LIN {X 0,Y 103.951,Z 742.341,A -85,B 0,C 180,E1 -28115.783,E2 -28115.783} C_VEL
LIN {X 0,Y 96.349,Z 750.933,A -85,B 0,C 180,E1 -28120.019,E2 -28120.019} C_VEL
LIN {X 0,Y 88.516,Z 758.718,A -85,B 0,C 180,E1 -28125.825,E2 -28125.825} C_VEL
LIN {X 0,Y 83.316,Z 763.333,A -85,B 0,C 180,E1 -28130.76,E2 -28130.76} C_VEL
LIN {X 0,Y 78.062,Z 767.663,A -85,B 0,C 180,E1 -28137.31,E2 -28137.31} C_VEL
LIN {X 0,Y 75.138,Z 769.96,A -85,B 0,C 180,E1 -28142.122,E2 -28142.122} C_VEL
LIN {X 0,Y 72.891,Z 771.823,A -85,B 0,C 180,E1 -28147.32,E2 -28147.32} C_VEL
LIN {X 0,Y 70.141,Z 774.222,A -85,B 0,C 180,E1 -28158.445,E2 -28158.445} C_VEL
LIN {X 0,Y 69.62,Z 774.834,A -85,B 0,C 180,E1 -28164.212,E2 -28164.212} C_VEL
LIN {X 0,Y 69.698,Z 775.05,A -85,B 0,C 180,E1 -28170.005,E2 -28170.005} C_VEL
LIN {X 0,Y 70.018,Z 774.825,A -85,B 0,C 180,E1 -28175.766,E2 -28175.766} C_VEL
LIN {X 0,Y 72.328,Z 773.205,A -85,B 0,C 180,E1 -28186.953,E2 -28186.953} C_VEL
LIN {X 0,Y 74.422,Z 771.801,A -85,B 0,C 180,E1 -28192.199,E2 -28192.199} C_VEL
LIN {X 0,Y 78.894,Z 768.873,A -85,B 0,C 180,E1 -28199.342,E2 -28199.342} C_VEL
LIN {X 0,Y 84.664,Z 764.918,A -85,B 0,C 180,E1 -28205.531,E2 -28205.531} C_VEL
LIN {X 0,Y 91.748,Z 759.838,A -85,B 0,C 180,E1 -28210.63,E2 -28210.63} C_VEL
LIN {X 0,Y 97.262,Z 756.003,A -85,B 0,C 180,E1 -28213.358,E2 -28213.358} C_VEL
LIN {X 0,Y 98.436,Z 756.44,A -85,B 0,C 180,E1 -28214.122,E2 -28214.122} C_VEL
LIN {X 0,Y 99.632,Z 757.554,A -85,B 0,C 180,E1 -28215.138,E2 -28215.138} C_VEL
LIN {X 0,Y 98.401,Z 756.23,A -85,B 0,C 180,E1 -28217.273,E2 -28217.273} C_VEL
LIN {X 0,Y 94.133,Z 751.514,A -85,B 0,C 180,E1 -28221.297,E2 -28221.297} C_VEL
LIN {X 0,Y 92.534,Z 750.794,A -85,B 0,C 180,E1 -28222.584,E2 -28222.584} C_VEL
LIN {X 0,Y 89.015,Z 750.077,A -85,B 0,C 180,E1 -28226.45,E2 -28226.45} C_VEL
LIN {X 0,Y 86.882,Z 747.385,A -85,B 0,C 180,E1 -28232.857,E2 -28232.857} C_VEL
LIN {X 0,Y 85.307,Z 746.912,A -85,B 0,C 180,E1 -28235.674,E2 -28235.674} C_VEL
LIN {X 0,Y 84.144,Z 745.468,A -85,B 0,C 180,E1 -28240.483,E2 -28240.483} C_VEL
LIN {X 0,Y 84.612,Z 743,A -85,B 0,C 180,E1 -28245.571,E2 -28245.571} C_VEL
LIN {X 0,Y 85.192,Z 740.288,A -85,B 0,C 180,E1 -28253.587,E2 -28253.587} C_VEL
LIN {X 0,Y 85.413,Z 739.646,A -85,B 0,C 180,E1 -28256.213,E2 -28256.213} C_VEL
LIN {X 0,Y 84.758,Z 739.885,A -85,B 0,C 180,E1 -28260.73,E2 -28260.73} C_VEL
LIN {X 0,Y 84.568,Z 740.192,A -85,B 0,C 180,E1 -28265.315,E2 -28265.315} C_VEL
LIN {X 0,Y 85.486,Z 739.643,A -85,B 0,C 180,E1 -28267.912,E2 -28267.912} C_VEL
LIN {X 0,Y 88.337,Z 737.785,A -85,B 0,C 180,E1 -28271.763,E2 -28271.763} C_VEL
LIN {X 0,Y 90.112,Z 736.61,A -85,B 0,C 180,E1 -28273.531,E2 -28273.531} C_VEL
LIN {X 0,Y 92.574,Z 734.85,A -85,B 0,C 180,E1 -28275.41,E2 -28275.41} C_VEL
LIN {X 0,Y 97.676,Z 731.683,A -85,B 0,C 180,E1 -28279.541,E2 -28279.541} C_VEL
LIN {X 0,Y 102.495,Z 728.307,A -85,B 0,C 180,E1 -28282.156,E2 -28282.156} C_VEL
LIN {X 0,Y 111.157,Z 722.092,A -85,B 0,C 180,E1 -28286.269,E2 -28286.269} C_VEL
LIN {X 0,Y 113.724,Z 720.096,A -85,B 0,C 180,E1 -28287.244,E2 -28287.244} C_VEL
LIN {X 0,Y 113.59,Z 721.326,A -85,B 0,C 180,E1 -28288.149,E2 -28288.149} C_VEL
LIN {X 0,Y 106.442,Z 731.795,A -85,B 0,C 180,E1 -28290.863,E2 -28290.863} C_VEL
LIN {X 0,Y 99.593,Z 740.264,A -85,B 0,C 180,E1 -28293.983,E2 -28293.983} C_VEL
LIN {X 0,Y 91.701,Z 748.632,A -85,B 0,C 180,E1 -28298.418,E2 -28298.418} C_VEL
LIN {X 0,Y 85.822,Z 754.124,A -85,B 0,C 180,E1 -28302.517,E2 -28302.517} C_VEL
LIN {X 0,Y 79.072,Z 759.618,A -85,B 0,C 180,E1 -28308.189,E2 -28308.189} C_VEL
LIN {X 0,Y 73.326,Z 763.919,A -85,B 0,C 180,E1 -28314.889,E2 -28314.889} C_VEL
LIN {X 0,Y 70.064,Z 766.192,A -85,B 0,C 180,E1 -28319.892,E2 -28319.892} C_VEL
LIN {X 0,Y 67.35,Z 768.037,A -85,B 0,C 180,E1 -28325.324,E2 -28325.324} C_VEL
LIN {X 0,Y 65.246,Z 769.422,A -85,B 0,C 180,E1 -28331.141,E2 -28331.141} C_VEL
LIN {X 0,Y 62.947,Z 771.009,A -85,B 0,C 180,E1 -28343.584,E2 -28343.584} C_VEL
LIN {X 0,Y 62.722,Z 771.232,A -85,B 0,C 180,E1 -28349.994,E2 -28349.994} C_VEL
LIN {X 0,Y 62.94,Z 771.037,A -85,B 0,C 180,E1 -28356.405,E2 -28356.405} C_VEL
LIN {X 0,Y 65.24,Z 769.487,A -85,B 0,C 180,E1 -28368.849,E2 -28368.849} C_VEL
LIN {X 0,Y 67.334,Z 768.13,A -85,B 0,C 180,E1 -28374.671,E2 -28374.671} C_VEL
LIN {X 0,Y 71.588,Z 765.258,A -85,B 0,C 180,E1 -28382.674,E2 -28382.674} C_VEL
LIN {X 0,Y 76.942,Z 761.361,A -85,B 0,C 180,E1 -28389.74,E2 -28389.74} C_VEL
LIN {X 0,Y 83.405,Z 756.332,A -85,B 0,C 180,E1 -28395.738,E2 -28395.738} C_VEL
LIN {X 0,Y 90.529,Z 749.996,A -85,B 0,C 180,E1 -28400.918,E2 -28400.918} C_VEL
LIN {X 0,Y 97.95,Z 742.366,A -85,B 0,C 180,E1 -28405.233,E2 -28405.233} C_VEL
LIN {X 0,Y 104.986,Z 733.989,A -85,B 0,C 180,E1 -28408.589,E2 -28408.589} C_VEL
LIN {X 0,Y 112.075,Z 724.121,A -85,B 0,C 180,E1 -28411.384,E2 -28411.384} C_VEL
LIN {X 0,Y 118.662,Z 713.001,A -85,B 0,C 180,E1 -28413.604,E2 -28413.604} C_VEL
LIN {X 0,Y 123.869,Z 702.096,A -85,B 0,C 180,E1 -28415.194,E2 -28415.194} C_VEL
LIN {X 0,Y 128.403,Z 690.023,A -85,B 0,C 180,E1 -28416.453,E2 -28416.453} C_VEL
LIN {X 0,Y 131.881,Z 677.141,A -85,B 0,C 180,E1 -28417.41,E2 -28417.41} C_VEL
LIN {X 0,Y 134.056,Z 664.506,A -85,B 0,C 180,E1 -28418.006,E2 -28418.006} C_VEL
LIN {X 0,Y 134.924,Z 656.338,A -85,B 0,C 180,E1 -28418.309,E2 -28418.309} C_VEL
LIN {X 0,Y 132.782,Z 650.972,A -85,B 0,C 180,E1 -28421.683,E2 -28421.683} C_VEL
LIN {X 0,Y 131.13,Z 647.298,A -85,B 0,C 180,E1 -28424.778,E2 -28424.778} C_VEL
LIN {X 0,Y 129.8,Z 644.377,A -85,B 0,C 180,E1 -28427.888,E2 -28427.888} C_VEL
LIN {X 0,Y 128.772,Z 641.836,A -85,B 0,C 180,E1 -28431.17,E2 -28431.17} C_VEL
LIN {X 0,Y 127.754,Z 638.207,A -85,B 0,C 180,E1 -28440,E2 -28440} C_VEL
LIN {X 0,Y 128.97,Z 642.375,A -85,B 0,C 180,E1 -28449.211,E2 -28449.211} C_VEL
LIN {X 0,Y 130.645,Z 646.22,A -85,B 0,C 180,E1 -28453.811,E2 -28453.811} C_VEL
LIN {X 0,Y 132.545,Z 650.385,A -85,B 0,C 180,E1 -28457.537,E2 -28457.537} C_VEL
LIN {X 0,Y 133.588,Z 653.257,A -85,B 0,C 180,E1 -28459.346,E2 -28459.346} C_VEL
LIN {X 0,Y 134.794,Z 657.853,A -85,B 0,C 180,E1 -28461.406,E2 -28461.406} C_VEL
LIN {X 0,Y 132.887,Z 673.229,A -85,B 0,C 180,E1 -28461.953,E2 -28461.953} C_VEL
LIN {X 0,Y 129.998,Z 686.389,A -85,B 0,C 180,E1 -28462.692,E2 -28462.692} C_VEL
LIN {X 0,Y 125.715,Z 699.337,A -85,B 0,C 180,E1 -28463.741,E2 -28463.741} C_VEL
LIN {X 0,Y 120.339,Z 711.572,A -85,B 0,C 180,E1 -28465.154,E2 -28465.154} C_VEL
LIN {X 0,Y 114.322,Z 722.478,A -85,B 0,C 180,E1 -28466.959,E2 -28466.959} C_VEL
LIN {X 0,Y 107.009,Z 733.323,A -85,B 0,C 180,E1 -28469.524,E2 -28469.524} C_VEL
LIN {X 0,Y 99.949,Z 742.138,A -85,B 0,C 180,E1 -28472.465,E2 -28472.465} C_VEL
LIN {X 0,Y 91.931,Z 750.73,A -85,B 0,C 180,E1 -28476.617,E2 -28476.617} C_VEL
LIN {X 0,Y 84.142,Z 757.985,A -85,B 0,C 180,E1 -28481.928,E2 -28481.928} C_VEL
LIN {X 0,Y 77.939,Z 763.129,A -85,B 0,C 180,E1 -28487.452,E2 -28487.452} C_VEL
LIN {X 0,Y 72.171,Z 767.458,A -85,B 0,C 180,E1 -28494.254,E2 -28494.254} C_VEL
LIN {X 0,Y 68.92,Z 769.755,A -85,B 0,C 180,E1 -28499.351,E2 -28499.351} C_VEL
LIN {X 0,Y 66.352,Z 771.617,A -85,B 0,C 180,E1 -28504.939,E2 -28504.939} C_VEL
LIN {X 0,Y 64.452,Z 773.016,A -85,B 0,C 180,E1 -28510.912,E2 -28510.912} C_VEL
LIN {X 0,Y 63.176,Z 774.017,A -85,B 0,C 180,E1 -28517.151,E2 -28517.151} C_VEL
LIN {X 0,Y 62.555,Z 774.629,A -85,B 0,C 180,E1 -28523.555,E2 -28523.555} C_VEL
LIN {X 0,Y 62.607,Z 774.846,A -85,B 0,C 180,E1 -28530.006,E2 -28530.006} C_VEL
LIN {X 0,Y 62.958,Z 774.62,A -85,B 0,C 180,E1 -28536.415,E2 -28536.415} C_VEL
LIN {X 0,Y 65.591,Z 773.001,A -85,B 0,C 180,E1 -28548.756,E2 -28548.756} C_VEL
LIN {X 0,Y 67.928,Z 771.596,A -85,B 0,C 180,E1 -28554.453,E2 -28554.453} C_VEL
LIN {X 0,Y 72.809,Z 768.668,A -85,B 0,C 180,E1 -28562.071,E2 -28562.071} C_VEL
LIN {X 0,Y 79.017,Z 764.713,A -85,B 0,C 180,E1 -28568.512,E2 -28568.512} C_VEL
LIN {X 0,Y 86.479,Z 759.632,A -85,B 0,C 180,E1 -28573.697,E2 -28573.697} C_VEL
LIN {X 0,Y 91.24,Z 756.158,A -85,B 0,C 180,E1 -28576.112,E2 -28576.112} C_VEL
LIN {X 0,Y 87.932,Z 754.779,A -85,B 0,C 180,E1 -28580.253,E2 -28580.253} C_VEL
LIN {X 0,Y 84.169,Z 754.131,A -85,B 0,C 180,E1 -28584.233,E2 -28584.233} C_VEL
LIN {X 0,Y 80.136,Z 751.193,A -85,B 0,C 180,E1 -28593.992,E2 -28593.992} C_VEL
LIN {X 0,Y 78.65,Z 749.984,A -85,B 0,C 180,E1 -28599.058,E2 -28599.058} C_VEL
LIN {X 0,Y 79.024,Z 746.684,A -85,B 0,C 180,E1 -28608.06,E2 -28608.06} C_VEL
LIN {X 0,Y 83.57,Z 741.075,A -85,B 0,C 180,E1 -28624.824,E2 -28624.824} C_VEL
LIN {X 0,Y 85.486,Z 739.643,A -85,B 0,C 180,E1 -28627.912,E2 -28627.912} C_VEL
LIN {X 0,Y 87.027,Z 738.869,A -85,B 0,C 180,E1 -28631.283,E2 -28631.283} C_VEL
LIN {X 0,Y 90.368,Z 738.328,A -85,B 0,C 180,E1 -28638.799,E2 -28638.799} C_VEL
LIN {X 0,Y 92.458,Z 737.403,A -85,B 0,C 180,E1 -28640.822,E2 -28640.822} C_VEL
LIN {X 0,Y 96.855,Z 734.883,A -85,B 0,C 180,E1 -28643.522,E2 -28643.522} C_VEL
LIN {X 0,Y 103.773,Z 730.418,A -85,B 0,C 180,E1 -28646.551,E2 -28646.551} C_VEL
LIN {X 0,Y 102.975,Z 732.004,A -85,B 0,C 180,E1 -28647.464,E2 -28647.464} C_VEL
LIN {X 0,Y 95.662,Z 740.618,A -85,B 0,C 180,E1 -28650.519,E2 -28650.519} C_VEL
LIN {X 0,Y 88.192,Z 748.173,A -85,B 0,C 180,E1 -28654.361,E2 -28654.361} C_VEL
LIN {X 0,Y 81.191,Z 754.331,A -85,B 0,C 180,E1 -28658.82,E2 -28658.82} C_VEL
LIN {X 0,Y 73.933,Z 759.824,A -85,B 0,C 180,E1 -28664.519,E2 -28664.519} C_VEL
LIN {X 0,Y 67.626,Z 764.125,A -85,B 0,C 180,E1 -28671.418,E2 -28671.418} C_VEL
LIN {X 0,Y 64.009,Z 766.398,A -85,B 0,C 180,E1 -28676.696,E2 -28676.696} C_VEL
LIN {X 0,Y 60.978,Z 768.242,A -85,B 0,C 180,E1 -28682.541,E2 -28682.541} C_VEL
LIN {X 0,Y 58.576,Z 769.627,A -85,B 0,C 180,E1 -28688.897,E2 -28688.897} C_VEL
LIN {X 0,Y 55.914,Z 771.214,A -85,B 0,C 180,E1 -28702.773,E2 -28702.773} C_VEL
LIN {X 0,Y 55.649,Z 771.436,A -85,B 0,C 180,E1 -28709.993,E2 -28709.993} C_VEL
LIN {X 0,Y 55.908,Z 771.241,A -85,B 0,C 180,E1 -28717.215,E2 -28717.215} C_VEL
LIN {X 0,Y 58.569,Z 769.691,A -85,B 0,C 180,E1 -28731.092,E2 -28731.092} C_VEL
LIN {X 0,Y 60.961,Z 768.334,A -85,B 0,C 180,E1 -28737.454,E2 -28737.454} C_VEL
LIN {X 0,Y 65.72,Z 765.462,A -85,B 0,C 180,E1 -28746.019,E2 -28746.019} C_VEL
LIN {X 0,Y 71.623,Z 761.565,A -85,B 0,C 180,E1 -28753.376,E2 -28753.376} C_VEL
LIN {X 0,Y 78.616,Z 756.535,A -85,B 0,C 180,E1 -28759.445,E2 -28759.445} C_VEL
LIN {X 0,Y 86.231,Z 750.199,A -85,B 0,C 180,E1 -28764.582,E2 -28764.582} C_VEL
LIN {X 0,Y 94.363,Z 742.273,A -85,B 0,C 180,E1 -28768.918,E2 -28768.918} C_VEL
LIN {X 0,Y 102.93,Z 732.412,A -85,B 0,C 180,E1 -28772.569,E2 -28772.569} C_VEL
LIN {X 0,Y 110.366,Z 722.044,A -85,B 0,C 180,E1 -28775.143,E2 -28775.143} C_VEL
LIN {X 0,Y 117.211,Z 710.357,A -85,B 0,C 180,E1 -28777.195,E2 -28777.195} C_VEL
LIN {X 0,Y 122.573,Z 698.847,A -85,B 0,C 180,E1 -28778.591,E2 -28778.591} C_VEL
LIN {X 0,Y 126.995,Z 686.165,A -85,B 0,C 180,E1 -28779.743,E2 -28779.743} C_VEL
LIN {X 0,Y 130.237,Z 673.11,A -85,B 0,C 180,E1 -28780.514,E2 -28780.514} C_VEL
LIN {X 0,Y 132.088,Z 659.976,A -85,B 0,C 180,E1 -28781.072,E2 -28781.072} C_VEL
LIN {X 0,Y 130.016,Z 654.54,A -85,B 0,C 180,E1 -28785.097,E2 -28785.097} C_VEL
LIN {X 0,Y 128.555,Z 651.088,A -85,B 0,C 180,E1 -28788.769,E2 -28788.769} C_VEL
LIN {X 0,Y 127.631,Z 648.651,A -85,B 0,C 180,E1 -28792.087,E2 -28792.087} C_VEL
LIN {X 0,Y 126.869,Z 645.407,A -85,B 0,C 180,E1 -28800,E2 -28800} C_VEL
LIN {X 0,Y 127.846,Z 649.203,A -85,B 0,C 180,E1 -28808.437,E2 -28808.437} C_VEL
LIN {X 0,Y 129.208,Z 652.693,A -85,B 0,C 180,E1 -28812.666,E2 -28812.666} C_VEL
LIN {X 0,Y 130.912,Z 656.842,A -85,B 0,C 180,E1 -28816.407,E2 -28816.407} C_VEL
LIN {X 0,Y 131.779,Z 659.786,A -85,B 0,C 180,E1 -28818.135,E2 -28818.135} C_VEL
LIN {X 0,Y 132.019,Z 660.871,A -85,B 0,C 180,E1 -28818.627,E2 -28818.627} C_VEL
LIN {X 0,Y 129.975,Z 675.524,A -85,B 0,C 180,E1 -28819.181,E2 -28819.181} C_VEL
LIN {X 0,Y 127.004,Z 687.602,A -85,B 0,C 180,E1 -28819.836,E2 -28819.836} C_VEL
LIN {X 0,Y 122.977,Z 699.263,A -85,B 0,C 180,E1 -28820.722,E2 -28820.722} C_VEL
LIN {X 0,Y 117.495,Z 711.372,A -85,B 0,C 180,E1 -28822.017,E2 -28822.017} C_VEL
LIN {X 0,Y 111.288,Z 722.278,A -85,B 0,C 180,E1 -28823.704,E2 -28823.704} C_VEL
LIN {X 0,Y 103.691,Z 733.121,A -85,B 0,C 180,E1 -28826.104,E2 -28826.104} C_VEL
LIN {X 0,Y 96.311,Z 741.935,A -85,B 0,C 180,E1 -28828.885,E2 -28828.885} C_VEL
LIN {X 0,Y 87.864,Z 750.526,A -85,B 0,C 180,E1 -28832.883,E2 -28832.883} C_VEL
LIN {X 0,Y 80.011,Z 757.409,A -85,B 0,C 180,E1 -28837.771,E2 -28837.771} C_VEL
LIN {X 0,Y 72.858,Z 762.925,A -85,B 0,C 180,E1 -28843.667,E2 -28843.667} C_VEL
LIN {X 0,Y 66.524,Z 767.254,A -85,B 0,C 180,E1 -28850.67,E2 -28850.67} C_VEL
LIN {X 0,Y 62.9,Z 769.551,A -85,B 0,C 180,E1 -28856.044,E2 -28856.044} C_VEL
LIN {X 0,Y 59.955,Z 771.412,A -85,B 0,C 180,E1 -28862.045,E2 -28862.045} C_VEL
LIN {X 0,Y 57.761,Z 772.811,A -85,B 0,C 180,E1 -28868.598,E2 -28868.598} C_VEL
LIN {X 0,Y 56.265,Z 773.812,A -85,B 0,C 180,E1 -28875.54,E2 -28875.54} C_VEL
LIN {X 0,Y 55.512,Z 774.425,A -85,B 0,C 180,E1 -28882.733,E2 -28882.733} C_VEL
LIN {X 0,Y 55.506,Z 774.641,A -85,B 0,C 180,E1 -28890.007,E2 -28890.007} C_VEL
LIN {X 0,Y 55.927,Z 774.416,A -85,B 0,C 180,E1 -28897.226,E2 -28897.226} C_VEL
LIN {X 0,Y 58.92,Z 772.796,A -85,B 0,C 180,E1 -28910.974,E2 -28910.974} C_VEL
LIN {X 0,Y 61.543,Z 771.391,A -85,B 0,C 180,E1 -28917.186,E2 -28917.186} C_VEL
LIN {X 0,Y 66.904,Z 768.463,A -85,B 0,C 180,E1 -28925.299,E2 -28925.299} C_VEL
LIN {X 0,Y 73.602,Z 764.507,A -85,B 0,C 180,E1 -28931.951,E2 -28931.951} C_VEL
LIN {X 0,Y 82.094,Z 759.017,A -85,B 0,C 180,E1 -28937.455,E2 -28937.455} C_VEL
LIN {X 0,Y 81.907,Z 758.248,A -85,B 0,C 180,E1 -28938.913,E2 -28938.913} C_VEL
LIN {X 0,Y 79.297,Z 757.85,A -85,B 0,C 180,E1 -28941.655,E2 -28941.655} C_VEL
LIN {X 0,Y 73.007,Z 754.1,A -85,B 0,C 180,E1 -28957.353,E2 -28957.353} C_VEL
LIN {X 0,Y 73.257,Z 750.666,A -85,B 0,C 180,E1 -28968.938,E2 -28968.938} C_VEL
LIN {X 0,Y 77.803,Z 745.904,A -85,B 0,C 180,E1 -28985.183,E2 -28985.183} C_VEL
LIN {X 0,Y 84.369,Z 742.026,A -85,B 0,C 180,E1 -28994.472,E2 -28994.472} C_VEL
LIN {X 0,Y 86.619,Z 740.762,A -85,B 0,C 180,E1 -28996.501,E2 -28996.501} C_VEL
LIN {X 0,Y 89.295,Z 739.089,A -85,B 0,C 180,E1 -28998.35,E2 -28998.35} C_VEL
LIN {X 0,Y 92.458,Z 737.403,A -85,B 0,C 180,E1 -29000.822,E2 -29000.822} C_VEL
LIN {X 0,Y 93.19,Z 737.288,A -85,B 0,C 180,E1 -29001.855,E2 -29001.855} C_VEL
LIN {X 0,Y 93.192,Z 738.159,A -85,B 0,C 180,E1 -29003.471,E2 -29003.471} C_VEL
LIN {X 0,Y 92.186,Z 740.039,A -85,B 0,C 180,E1 -29005.254,E2 -29005.254} C_VEL
LIN {X 0,Y 90.512,Z 742.304,A -85,B 0,C 180,E1 -29006.911,E2 -29006.911} C_VEL
LIN {X 0,Y 86.442,Z 746.532,A -85,B 0,C 180,E1 -29009.368,E2 -29009.368} C_VEL
LIN {X 0,Y 79.905,Z 752.231,A -85,B 0,C 180,E1 -29012.928,E2 -29012.928} C_VEL
LIN {X 0,Y 76.543,Z 754.826,A -85,B 0,C 180,E1 -29014.936,E2 -29014.936} C_VEL
LIN {X 0,Y 69.143,Z 760.03,A -85,B 0,C 180,E1 -29020.322,E2 -29020.322} C_VEL
LIN {X 0,Y 62.218,Z 764.331,A -85,B 0,C 180,E1 -29027.325,E2 -29027.325} C_VEL
LIN {X 0,Y 58.202,Z 766.603,A -85,B 0,C 180,E1 -29032.853,E2 -29032.853} C_VEL
LIN {X 0,Y 54.761,Z 768.448,A -85,B 0,C 180,E1 -29039.105,E2 -29039.105} C_VEL
LIN {X 0,Y 50.04,Z 770.816,A -85,B 0,C 180,E1 -29053.679,E2 -29053.679} C_VEL
LIN {X 0,Y 48.878,Z 771.418,A -85,B 0,C 180,E1 -29061.726,E2 -29061.726} C_VEL
LIN {X 0,Y 48.565,Z 771.64,A -85,B 0,C 180,E1 -29069.993,E2 -29069.993} C_VEL
LIN {X 0,Y 48.874,Z 771.445,A -85,B 0,C 180,E1 -29078.26,E2 -29078.26} C_VEL
LIN {X 0,Y 50.037,Z 770.861,A -85,B 0,C 180,E1 -29086.307,E2 -29086.307} C_VEL
LIN {X 0,Y 54.743,Z 768.539,A -85,B 0,C 180,E1 -29100.891,E2 -29100.891} C_VEL
LIN {X 0,Y 60.121,Z 765.666,A -85,B 0,C 180,E1 -29110.003,E2 -29110.003} C_VEL
LIN {X 0,Y 66.641,Z 761.769,A -85,B 0,C 180,E1 -29117.572,E2 -29117.572} C_VEL
LIN {X 0,Y 74.199,Z 756.738,A -85,B 0,C 180,E1 -29123.612,E2 -29123.612} C_VEL
LIN {X 0,Y 82.322,Z 750.401,A -85,B 0,C 180,E1 -29128.609,E2 -29128.609} C_VEL
LIN {X 0,Y 90.9,Z 742.475,A -85,B 0,C 180,E1 -29132.755,E2 -29132.755} C_VEL
LIN {X 0,Y 98.346,Z 734.392,A -85,B 0,C 180,E1 -29135.654,E2 -29135.654} C_VEL
LIN {X 0,Y 106.021,Z 724.523,A -85,B 0,C 180,E1 -29138.121,E2 -29138.121} C_VEL
LIN {X 0,Y 113.075,Z 713.401,A -85,B 0,C 180,E1 -29140.053,E2 -29140.053} C_VEL
LIN {X 0,Y 118.627,Z 702.493,A -85,B 0,C 180,E1 -29141.414,E2 -29141.414} C_VEL
LIN {X 0,Y 123.368,Z 690.583,A -85,B 0,C 180,E1 -29142.483,E2 -29142.483} C_VEL
LIN {X 0,Y 127.027,Z 677.928,A -85,B 0,C 180,E1 -29143.295,E2 -29143.295} C_VEL
LIN {X 0,Y 129.382,Z 665.138,A -85,B 0,C 180,E1 -29143.828,E2 -29143.828} C_VEL
LIN {X 0,Y 129.499,Z 663.904,A -85,B 0,C 180,E1 -29143.937,E2 -29143.937} C_VEL
LIN {X 0,Y 128.047,Z 659.755,A -85,B 0,C 180,E1 -29147.519,E2 -29147.519} C_VEL
LIN {X 0,Y 127.06,Z 657.075,A -85,B 0,C 180,E1 -29150.649,E2 -29150.649} C_VEL
LIN {X 0,Y 126.571,Z 655.511,A -85,B 0,C 180,E1 -29152.823,E2 -29152.823} C_VEL
LIN {X 0,Y 125.989,Z 652.578,A -85,B 0,C 180,E1 -29160,E2 -29160} C_VEL
LIN {X 0,Y 126.735,Z 655.923,A -85,B 0,C 180,E1 -29167.568,E2 -29167.568} C_VEL
LIN {X 0,Y 127.96,Z 659.546,A -85,B 0,C 180,E1 -29171.886,E2 -29171.886} C_VEL
LIN {X 0,Y 129.296,Z 663.177,A -85,B 0,C 180,E1 -29175.164,E2 -29175.164} C_VEL
LIN {X 0,Y 129.547,Z 664.051,A -85,B 0,C 180,E1 -29175.739,E2 -29175.739} C_VEL
LIN {X 0,Y 127.446,Z 677.023,A -85,B 0,C 180,E1 -29176.25,E2 -29176.25} C_VEL
LIN {X 0,Y 123.759,Z 690.696,A -85,B 0,C 180,E1 -29176.989,E2 -29176.989} C_VEL
LIN {X 0,Y 119.007,Z 702.96,A -85,B 0,C 180,E1 -29177.901,E2 -29177.901} C_VEL
LIN {X 0,Y 113.427,Z 714.111,A -85,B 0,C 180,E1 -29179.119,E2 -29179.119} C_VEL
LIN {X 0,Y 106.259,Z 725.604,A -85,B 0,C 180,E1 -29180.907,E2 -29180.907} C_VEL
LIN {X 0,Y 99.202,Z 734.859,A -85,B 0,C 180,E1 -29182.94,E2 -29182.94} C_VEL
LIN {X 0,Y 90.072,Z 744.795,A -85,B 0,C 180,E1 -29186.204,E2 -29186.204} C_VEL
LIN {X 0,Y 81.359,Z 752.797,A -85,B 0,C 180,E1 -29190.26,E2 -29190.26} C_VEL
LIN {X 0,Y 72.509,Z 759.682,A -85,B 0,C 180,E1 -29195.787,E2 -29195.787} C_VEL
LIN {X 0,Y 65.675,Z 764.306,A -85,B 0,C 180,E1 -29201.498,E2 -29201.498} C_VEL
LIN {X 0,Y 59.09,Z 768.271,A -85,B 0,C 180,E1 -29209.153,E2 -29209.153} C_VEL
LIN {X 0,Y 53.749,Z 771.206,A -85,B 0,C 180,E1 -29218.473,E2 -29218.473} C_VEL
LIN {X 0,Y 51.174,Z 772.605,A -85,B 0,C 180,E1 -29225.677,E2 -29225.677} C_VEL
LIN {X 0,Y 48.472,Z 774.22,A -85,B 0,C 180,E1 -29241.671,E2 -29241.671} C_VEL
LIN {X 0,Y 48.423,Z 774.437,A -85,B 0,C 180,E1 -29250.007,E2 -29250.007} C_VEL
LIN {X 0,Y 48.894,Z 774.211,A -85,B 0,C 180,E1 -29258.272,E2 -29258.272} C_VEL
LIN {X 0,Y 52.353,Z 772.591,A -85,B 0,C 180,E1 -29273.756,E2 -29273.756} C_VEL
LIN {X 0,Y 55.338,Z 771.186,A -85,B 0,C 180,E1 -29280.539,E2 -29280.539} C_VEL
LIN {X 0,Y 61.257,Z 768.257,A -85,B 0,C 180,E1 -29289.132,E2 -29289.132} C_VEL
LIN {X 0,Y 68.499,Z 764.302,A -85,B 0,C 180,E1 -29295.913,E2 -29295.913} C_VEL
LIN {X 0,Y 71.167,Z 762.715,A -85,B 0,C 180,E1 -29297.794,E2 -29297.794} C_VEL
LIN {X 0,Y 73.283,Z 760.996,A -85,B 0,C 180,E1 -29300.112,E2 -29300.112} C_VEL
LIN {X 0,Y 67.223,Z 757.885,A -85,B 0,C 180,E1 -29315.28,E2 -29315.28} C_VEL
LIN {X 0,Y 66.509,Z 756.407,A -85,B 0,C 180,E1 -29322.01,E2 -29322.01} C_VEL
LIN {X 0,Y 67.886,Z 753.396,A -85,B 0,C 180,E1 -29334.058,E2 -29334.058} C_VEL
LIN {X 0,Y 74.886,Z 748.686,A -85,B 0,C 180,E1 -29350.819,E2 -29350.819} C_VEL
LIN {X 0,Y 81.479,Z 745.492,A -85,B 0,C 180,E1 -29358.399,E2 -29358.399} C_VEL
LIN {X 0,Y 86.079,Z 743.1,A -85,B 0,C 180,E1 -29361.556,E2 -29361.556} C_VEL
LIN {X 0,Y 92.54,Z 740.012,A -85,B 0,C 180,E1 -29365.709,E2 -29365.709} C_VEL
LIN {X 0,Y 91.459,Z 741.624,A -85,B 0,C 180,E1 -29367.043,E2 -29367.043} C_VEL
LIN {X 0,Y 82.367,Z 750.135,A -85,B 0,C 180,E1 -29371.425,E2 -29371.425} C_VEL
LIN {X 0,Y 76.543,Z 754.826,A -85,B 0,C 180,E1 -29374.936,E2 -29374.936} C_VEL
LIN {X 0,Y 72.253,Z 757.693,A -85,B 0,C 180,E1 -29377.183,E2 -29377.183} C_VEL
LIN {X 0,Y 64.153,Z 761.892,A -85,B 0,C 180,E1 -29380.444,E2 -29380.444} C_VEL
LIN {X 0,Y 56.103,Z 765.387,A -85,B 0,C 180,E1 -29384.84,E2 -29384.84} C_VEL
LIN {X 0,Y 52.11,Z 767.076,A -85,B 0,C 180,E1 -29389.086,E2 -29389.086} C_VEL
LIN {X 0,Y 48.799,Z 768.654,A -85,B 0,C 180,E1 -29394.816,E2 -29394.816} C_VEL
LIN {X 0,Y 43.276,Z 771.021,A -85,B 0,C 180,E1 -29411.038,E2 -29411.038} C_VEL
LIN {X 0,Y 41.882,Z 771.623,A -85,B 0,C 180,E1 -29420.331,E2 -29420.331} C_VEL
LIN {X 0,Y 41.469,Z 771.845,A -85,B 0,C 180,E1 -29429.991,E2 -29429.991} C_VEL
LIN {X 0,Y 41.877,Z 771.649,A -85,B 0,C 180,E1 -29439.652,E2 -29439.652} C_VEL
LIN {X 0,Y 43.271,Z 771.065,A -85,B 0,C 180,E1 -29448.946,E2 -29448.946} C_VEL
LIN {X 0,Y 48.78,Z 768.743,A -85,B 0,C 180,E1 -29465.182,E2 -29465.182} C_VEL
LIN {X 0,Y 54.872,Z 765.869,A -85,B 0,C 180,E1 -29474.775,E2 -29474.775} C_VEL
LIN {X 0,Y 62.076,Z 761.972,A -85,B 0,C 180,E1 -29482.411,E2 -29482.411} C_VEL
LIN {X 0,Y 70.223,Z 756.941,A -85,B 0,C 180,E1 -29488.276,E2 -29488.276} C_VEL
LIN {X 0,Y 78.862,Z 750.604,A -85,B 0,C 180,E1 -29493.011,E2 -29493.011} C_VEL
LIN {X 0,Y 87.873,Z 742.678,A -85,B 0,C 180,E1 -29496.879,E2 -29496.879} C_VEL
LIN {X 0,Y 97.212,Z 732.815,A -85,B 0,C 180,E1 -29500.013,E2 -29500.013} C_VEL
LIN {X 0,Y 105.199,Z 722.445,A -85,B 0,C 180,E1 -29502.163,E2 -29502.163} C_VEL
LIN {X 0,Y 112.476,Z 710.757,A -85,B 0,C 180,E1 -29503.869,E2 -29503.869} C_VEL
LIN {X 0,Y 117.921,Z 699.778,A -85,B 0,C 180,E1 -29504.95,E2 -29504.95} C_VEL
LIN {X 0,Y 122.315,Z 688.136,A -85,B 0,C 180,E1 -29505.855,E2 -29505.855} C_VEL
LIN {X 0,Y 125.98,Z 674.558,A -85,B 0,C 180,E1 -29506.545,E2 -29506.545} C_VEL
LIN {X 0,Y 127.16,Z 668.118,A -85,B 0,C 180,E1 -29506.861,E2 -29506.861} C_VEL
LIN {X 0,Y 126.024,Z 664.182,A -85,B 0,C 180,E1 -29510.976,E2 -29510.976} C_VEL
LIN {X 0,Y 125.461,Z 662.197,A -85,B 0,C 180,E1 -29513.971,E2 -29513.971} C_VEL
LIN {X 0,Y 125.114,Z 659.701,A -85,B 0,C 180,E1 -29520,E2 -29520} C_VEL
LIN {X 0,Y 125.67,Z 662.816,A -85,B 0,C 180,E1 -29526.825,E2 -29526.825} C_VEL
LIN {X 0,Y 126.54,Z 665.882,A -85,B 0,C 180,E1 -29530.601,E2 -29530.601} C_VEL
LIN {X 0,Y 127.22,Z 668.096,A -85,B 0,C 180,E1 -29532.766,E2 -29532.766} C_VEL
LIN {X 0,Y 124.688,Z 680.934,A -85,B 0,C 180,E1 -29533.3,E2 -29533.3} C_VEL
LIN {X 0,Y 120.47,Z 694.404,A -85,B 0,C 180,E1 -29534.025,E2 -29534.025} C_VEL
LIN {X 0,Y 115.424,Z 706.15,A -85,B 0,C 180,E1 -29534.863,E2 -29534.863} C_VEL
LIN {X 0,Y 108.835,Z 718.048,A -85,B 0,C 180,E1 -29536.162,E2 -29536.162} C_VEL
LIN {X 0,Y 101.483,Z 728.661,A -85,B 0,C 180,E1 -29537.794,E2 -29537.794} C_VEL
LIN {X 0,Y 93.478,Z 738.235,A -85,B 0,C 180,E1 -29539.996,E2 -29539.996} C_VEL
LIN {X 0,Y 84.076,Z 747.448,A -85,B 0,C 180,E1 -29543.158,E2 -29543.158} C_VEL
LIN {X 0,Y 75.049,Z 754.866,A -85,B 0,C 180,E1 -29547.185,E2 -29547.185} C_VEL
LIN {X 0,Y 66.558,Z 760.827,A -85,B 0,C 180,E1 -29552.367,E2 -29552.367} C_VEL
LIN {X 0,Y 58.633,Z 765.536,A -85,B 0,C 180,E1 -29558.83,E2 -29558.83} C_VEL
LIN {X 0,Y 51.715,Z 769.143,A -85,B 0,C 180,E1 -29567.205,E2 -29567.205} C_VEL
LIN {X 0,Y 47.809,Z 771.001,A -85,B 0,C 180,E1 -29573.994,E2 -29573.994} C_VEL
LIN {X 0,Y 42.607,Z 773.401,A -85,B 0,C 180,E1 -29590.746,E2 -29590.746} C_VEL
LIN {X 0,Y 41.446,Z 774.015,A -85,B 0,C 180,E1 -29600.246,E2 -29600.246} C_VEL
LIN {X 0,Y 41.323,Z 774.232,A -85,B 0,C 180,E1 -29610.009,E2 -29610.009} C_VEL
LIN {X 0,Y 41.897,Z 774.006,A -85,B 0,C 180,E1 -29619.665,E2 -29619.665} C_VEL
LIN {X 0,Y 45.954,Z 772.386,A -85,B 0,C 180,E1 -29637.319,E2 -29637.319} C_VEL
LIN {X 0,Y 49.356,Z 770.981,A -85,B 0,C 180,E1 -29644.729,E2 -29644.729} C_VEL
LIN {X 0,Y 55.945,Z 768.052,A -85,B 0,C 180,E1 -29653.712,E2 -29653.712} C_VEL
LIN {X 0,Y 63.78,Z 764.097,A -85,B 0,C 180,E1 -29660.483,E2 -29660.483} C_VEL
LIN {X 0,Y 64.691,Z 763.049,A -85,B 0,C 180,E1 -29662.677,E2 -29662.677} C_VEL
LIN {X 0,Y 60.314,Z 760.1,A -85,B 0,C 180,E1 -29679.539,E2 -29679.539} C_VEL
LIN {X 0,Y 63.26,Z 755.793,A -85,B 0,C 180,E1 -29700.517,E2 -29700.517} C_VEL
LIN {X 0,Y 72.642,Z 751.304,A -85,B 0,C 180,E1 -29716.873,E2 -29716.873} C_VEL
LIN {X 0,Y 79.864,Z 748.328,A -85,B 0,C 180,E1 -29723.328,E2 -29723.328} C_VEL
LIN {X 0,Y 82.975,Z 746.872,A -85,B 0,C 180,E1 -29725.056,E2 -29725.056} C_VEL
LIN {X 0,Y 74.572,Z 753.72,A -85,B 0,C 180,E1 -29729.328,E2 -29729.328} C_VEL
LIN {X 0,Y 67.492,Z 758.547,A -85,B 0,C 180,E1 -29733.577,E2 -29733.577} C_VEL
LIN {X 0,Y 59.611,Z 763.234,A -85,B 0,C 180,E1 -29739.965,E2 -29739.965} C_VEL
LIN {X 0,Y 52.11,Z 767.076,A -85,B 0,C 180,E1 -29749.086,E2 -29749.086} C_VEL
LIN {X 0,Y 48.394,Z 768.608,A -85,B 0,C 180,E1 -29754.079,E2 -29754.079} C_VEL
LIN {X 0,Y 41.577,Z 770.487,A -85,B 0,C 180,E1 -29762.975,E2 -29762.975} C_VEL
LIN {X 0,Y 36.836,Z 771.507,A -85,B 0,C 180,E1 -29772.252,E2 -29772.252} C_VEL
LIN {X 0,Y 34.558,Z 771.956,A -85,B 0,C 180,E1 -29782.74,E2 -29782.74} C_VEL
LIN {X 0,Y 34.456,Z 771.943,A -85,B 0,C 180,E1 -29784.373,E2 -29784.373} C_VEL
LIN {X 0,Y 34.894,Z 771.854,A -85,B 0,C 180,E1 -29801.609,E2 -29801.609} C_VEL
LIN {X 0,Y 39.445,Z 770.304,A -85,B 0,C 180,E1 -29822.3,E2 -29822.3} C_VEL
LIN {X 0,Y 43.172,Z 768.947,A -85,B 0,C 180,E1 -29830.618,E2 -29830.618} C_VEL
LIN {X 0,Y 50.065,Z 766.074,A -85,B 0,C 180,E1 -29840.529,E2 -29840.529} C_VEL
LIN {X 0,Y 58.023,Z 762.175,A -85,B 0,C 180,E1 -29847.968,E2 -29847.968} C_VEL
LIN {X 0,Y 66.767,Z 757.144,A -85,B 0,C 180,E1 -29853.46,E2 -29853.46} C_VEL
LIN {X 0,Y 75.908,Z 750.806,A -85,B 0,C 180,E1 -29857.784,E2 -29857.784} C_VEL
LIN {X 0,Y 85.333,Z 742.88,A -85,B 0,C 180,E1 -29861.272,E2 -29861.272} C_VEL
LIN {X 0,Y 93.393,Z 734.796,A -85,B 0,C 180,E1 -29863.614,E2 -29863.614} C_VEL
LIN {X 0,Y 101.591,Z 724.925,A -85,B 0,C 180,E1 -29865.567,E2 -29865.567} C_VEL
LIN {X 0,Y 109.056,Z 713.801,A -85,B 0,C 180,E1 -29867.071,E2 -29867.071} C_VEL
LIN {X 0,Y 115.534,Z 701.578,A -85,B 0,C 180,E1 -29868.202,E2 -29868.202} C_VEL
LIN {X 0,Y 120.225,Z 690.015,A -85,B 0,C 180,E1 -29869.011,E2 -29869.011} C_VEL
LIN {X 0,Y 123.849,Z 677.648,A -85,B 0,C 180,E1 -29869.631,E2 -29869.631} C_VEL
LIN {X 0,Y 124.949,Z 672.595,A -85,B 0,C 180,E1 -29869.877,E2 -29869.877} C_VEL
LIN {X 0,Y 124.372,Z 669.364,A -85,B 0,C 180,E1 -29873.918,E2 -29873.918} C_VEL
LIN {X 0,Y 124.144,Z 666.891,A -85,B 0,C 180,E1 -29880,E2 -29880} C_VEL
LIN {X 0,Y 124.451,Z 669.656,A -85,B 0,C 180,E1 -29886.078,E2 -29886.078} C_VEL
LIN {X 0,Y 125.029,Z 672.639,A -85,B 0,C 180,E1 -29889.762,E2 -29889.762} C_VEL
LIN {X 0,Y 122.067,Z 685.002,A -85,B 0,C 180,E1 -29890.259,E2 -29890.259} C_VEL
LIN {X 0,Y 117.902,Z 696.935,A -85,B 0,C 180,E1 -29890.868,E2 -29890.868} C_VEL
LIN {X 0,Y 112.966,Z 707.605,A -85,B 0,C 180,E1 -29891.537,E2 -29891.537} C_VEL
LIN {X 0,Y 106.239,Z 719.141,A -85,B 0,C 180,E1 -29892.66,E2 -29892.66} C_VEL
LIN {X 0,Y 98.714,Z 729.531,A -85,B 0,C 180,E1 -29894.079,E2 -29894.079} C_VEL
LIN {X 0,Y 91.292,Z 738.033,A -85,B 0,C 180,E1 -29895.8,E2 -29895.8} C_VEL
LIN {X 0,Y 83.136,Z 745.874,A -85,B 0,C 180,E1 -29898.02,E2 -29898.02} C_VEL
LIN {X 0,Y 73.625,Z 753.541,A -85,B 0,C 180,E1 -29901.47,E2 -29901.47} C_VEL
LIN {X 0,Y 63.019,Z 760.622,A -85,B 0,C 180,E1 -29906.866,E2 -29906.866} C_VEL
LIN {X 0,Y 54.446,Z 765.331,A -85,B 0,C 180,E1 -29912.975,E2 -29912.975} C_VEL
LIN {X 0,Y 46.746,Z 768.938,A -85,B 0,C 180,E1 -29921.273,E2 -29921.273} C_VEL
LIN {X 0,Y 42.245,Z 770.796,A -85,B 0,C 180,E1 -29928.294,E2 -29928.294} C_VEL
LIN {X 0,Y 35.966,Z 773.197,A -85,B 0,C 180,E1 -29947.006,E2 -29947.006} C_VEL
LIN {X 0,Y 34.467,Z 773.81,A -85,B 0,C 180,E1 -29958.246,E2 -29958.246} C_VEL
LIN {X 0,Y 34.237,Z 774.028,A -85,B 0,C 180,E1 -29970.011,E2 -29970.011} C_VEL
LIN {X 0,Y 34.93,Z 773.802,A -85,B 0,C 180,E1 -29981.618,E2 -29981.618} C_VEL
LIN {X 0,Y 39.797,Z 772.181,A -85,B 0,C 180,E1 -30002.002,E2 -30002.002} C_VEL
LIN {X 0,Y 43.717,Z 770.776,A -85,B 0,C 180,E1 -30010.03,E2 -30010.03} C_VEL
LIN {X 0,Y 51.067,Z 767.848,A -85,B 0,C 180,E1 -30019.204,E2 -30019.204} C_VEL
LIN {X 0,Y 56.015,Z 765.607,A -85,B 0,C 180,E1 -30023.385,E2 -30023.385} C_VEL
LIN {X 0,Y 55.409,Z 764.325,A -85,B 0,C 180,E1 -30029.512,E2 -30029.512} C_VEL
LIN {X 0,Y 53.862,Z 762.066,A -85,B 0,C 180,E1 -30044.873,E2 -30044.873} C_VEL
LIN {X 0,Y 66.47,Z 755.323,A -85,B 0,C 180,E1 -30078.494,E2 -30078.494} C_VEL
LIN {X 0,Y 71.2,Z 753.712,A -85,B 0,C 180,E1 -30083.256,E2 -30083.256} C_VEL
LIN {X 0,Y 69.826,Z 754.951,A -85,B 0,C 180,E1 -30085.051,E2 -30085.051} C_VEL
LIN {X 0,Y 60.932,Z 760.441,A -85,B 0,C 180,E1 -30090.099,E2 -30090.099} C_VEL
LIN {X 0,Y 52.643,Z 764.744,A -85,B 0,C 180,E1 -30096.761,E2 -30096.761} C_VEL
LIN {X 0,Y 46.649,Z 767.412,A -85,B 0,C 180,E1 -30103.867,E2 -30103.867} C_VEL
LIN {X 0,Y 39.454,Z 770.242,A -85,B 0,C 180,E1 -30117.687,E2 -30117.687} C_VEL
LIN {X 0,Y 34.898,Z 771.828,A -85,B 0,C 180,E1 -30138.371,E2 -30138.371} C_VEL
LIN {X 0,Y 34.456,Z 771.943,A -85,B 0,C 180,E1 -30144.373,E2 -30144.373} C_VEL
LIN {X 0,Y 33.759,Z 772.041,A -85,B 0,C 180,E1 -30154.206,E2 -30154.206} C_VEL
LIN {X 0,Y 32.946,Z 771.869,A -85,B 0,C 180,E1 -30164.327,E2 -30164.327} C_VEL
LIN {X 0,Y 33.568,Z 770.764,A -85,B 0,C 180,E1 -30184.994,E2 -30184.994} C_VEL
LIN {X 0,Y 36.042,Z 769.794,A -85,B 0,C 180,E1 -30193.816,E2 -30193.816} C_VEL
LIN {X 0,Y 37.251,Z 769.385,A -85,B 0,C 180,E1 -30196.224,E2 -30196.224} C_VEL
LIN {X 0,Y 45.87,Z 766.278,A -85,B 0,C 180,E1 -30207.41,E2 -30207.41} C_VEL
LIN {X 0,Y 54.596,Z 762.379,A -85,B 0,C 180,E1 -30214.286,E2 -30214.286} C_VEL
LIN {X 0,Y 63.914,Z 757.347,A -85,B 0,C 180,E1 -30219.157,E2 -30219.157} C_VEL
LIN {X 0,Y 73.522,Z 751.008,A -85,B 0,C 180,E1 -30222.902,E2 -30222.902} C_VEL
LIN {X 0,Y 83.321,Z 743.083,A -85,B 0,C 180,E1 -30225.913,E2 -30225.913} C_VEL
LIN {X 0,Y 91.647,Z 734.997,A -85,B 0,C 180,E1 -30227.867,E2 -30227.867} C_VEL
LIN {X 0,Y 100.058,Z 725.127,A -85,B 0,C 180,E1 -30229.508,E2 -30229.508} C_VEL
LIN {X 0,Y 107.691,Z 714.001,A -85,B 0,C 180,E1 -30230.754,E2 -30230.754} C_VEL
LIN {X 0,Y 114.221,Z 701.929,A -85,B 0,C 180,E1 -30231.674,E2 -30231.674} C_VEL
LIN {X 0,Y 119.342,Z 689.44,A -85,B 0,C 180,E1 -30232.414,E2 -30232.414} C_VEL
LIN {X 0,Y 122.874,Z 677.379,A -85,B 0,C 180,E1 -30232.92,E2 -30232.92} C_VEL
LIN {X 0,Y 122.731,Z 675.561,A -85,B 0,C 180,E1 -30235.895,E2 -30235.895} C_VEL
LIN {X 0,Y 122.838,Z 674.013,A -85,B 0,C 180,E1 -30240,E2 -30240} C_VEL
LIN {X 0,Y 122.866,Z 676.271,A -85,B 0,C 180,E1 -30245.128,E2 -30245.128} C_VEL
LIN {X 0,Y 122.972,Z 677.344,A -85,B 0,C 180,E1 -30246.676,E2 -30246.676} C_VEL
LIN {X 0,Y 119.3,Z 690.059,A -85,B 0,C 180,E1 -30247.142,E2 -30247.142} C_VEL
LIN {X 0,Y 114.641,Z 701.595,A -85,B 0,C 180,E1 -30247.633,E2 -30247.633} C_VEL
LIN {X 0,Y 108.335,Z 713.51,A -85,B 0,C 180,E1 -30248.41,E2 -30248.41} C_VEL
LIN {X 0,Y 100.64,Z 725,A -85,B 0,C 180,E1 -30249.488,E2 -30249.488} C_VEL
LIN {X 0,Y 92.982,Z 734.252,A -85,B 0,C 180,E1 -30250.727,E2 -30250.727} C_VEL
LIN {X 0,Y 84.563,Z 742.696,A -85,B 0,C 180,E1 -30252.458,E2 -30252.458} C_VEL
LIN {X 0,Y 74.596,Z 750.949,A -85,B 0,C 180,E1 -30255.073,E2 -30255.073} C_VEL
LIN {X 0,Y 66.469,Z 756.591,A -85,B 0,C 180,E1 -30257.917,E2 -30257.917} C_VEL
LIN {X 0,Y 57.031,Z 762.108,A -85,B 0,C 180,E1 -30262.464,E2 -30262.464} C_VEL
LIN {X 0,Y 47.979,Z 766.435,A -85,B 0,C 180,E1 -30268.508,E2 -30268.508} C_VEL
LIN {X 0,Y 42.378,Z 768.733,A -85,B 0,C 180,E1 -30273.998,E2 -30273.998} C_VEL
LIN {X 0,Y 37.222,Z 770.591,A -85,B 0,C 180,E1 -30280.968,E2 -30280.968} C_VEL
LIN {X 0,Y 32.885,Z 771.99,A -85,B 0,C 180,E1 -30290.137,E2 -30290.137} C_VEL
LIN {X 0,Y 27.537,Z 773.605,A -85,B 0,C 180,E1 -30315.227,E2 -30315.227} C_VEL
LIN {X 0,Y 27.123,Z 773.823,A -85,B 0,C 180,E1 -30330.013,E2 -30330.013} C_VEL
LIN {X 0,Y 28.012,Z 773.597,A -85,B 0,C 180,E1 -30344.544,E2 -30344.544} C_VEL
LIN {X 0,Y 33.986,Z 771.976,A -85,B 0,C 180,E1 -30368.356,E2 -30368.356} C_VEL
LIN {X 0,Y 38.564,Z 770.571,A -85,B 0,C 180,E1 -30376.813,E2 -30376.813} C_VEL
LIN {X 0,Y 48.228,Z 767.039,A -85,B 0,C 180,E1 -30386.934,E2 -30386.934} C_VEL
LIN {X 0,Y 48.194,Z 766.333,A -85,B 0,C 180,E1 -30391.055,E2 -30391.055} C_VEL
LIN {X 0,Y 55.837,Z 760.313,A -85,B 0,C 180,E1 -30434.581,E2 -30434.581} C_VEL
LIN {X 0,Y 60.169,Z 758.955,A -85,B 0,C 180,E1 -30440.513,E2 -30440.513} C_VEL
LIN {X 0,Y 60.802,Z 758.96,A -85,B 0,C 180,E1 -30442.36,E2 -30442.36} C_VEL
LIN {X 0,Y 51.652,Z 763.646,A -85,B 0,C 180,E1 -30447.805,E2 -30447.805} C_VEL
LIN {X 0,Y 43.197,Z 767.219,A -85,B 0,C 180,E1 -30455.548,E2 -30455.548} C_VEL
LIN {X 0,Y 38.089,Z 769.064,A -85,B 0,C 180,E1 -30462.42,E2 -30462.42} C_VEL
LIN {X 0,Y 30.203,Z 771.431,A -85,B 0,C 180,E1 -30482.252,E2 -30482.252} C_VEL
LIN {X 0,Y 27.381,Z 772.154,A -85,B 0,C 180,E1 -30503.361,E2 -30503.361} C_VEL
LIN {X 0,Y 27.971,Z 772.058,A -85,B 0,C 180,E1 -30524.539,E2 -30524.539} C_VEL
LIN {X 0,Y 30.197,Z 771.474,A -85,B 0,C 180,E1 -30537.727,E2 -30537.727} C_VEL
LIN {X 0,Y 37.251,Z 769.385,A -85,B 0,C 180,E1 -30556.224,E2 -30556.224} C_VEL
LIN {X 0,Y 40.823,Z 768.136,A -85,B 0,C 180,E1 -30562.889,E2 -30562.889} C_VEL
LIN {X 0,Y 46.363,Z 765.536,A -85,B 0,C 180,E1 -30573.184,E2 -30573.184} C_VEL
LIN {X 0,Y 52.837,Z 762.244,A -85,B 0,C 180,E1 -30581.005,E2 -30581.005} C_VEL
LIN {X 0,Y 57.527,Z 759.812,A -85,B 0,C 180,E1 -30583.796,E2 -30583.796} C_VEL
LIN {X 0,Y 68.39,Z 753.462,A -85,B 0,C 180,E1 -30587.462,E2 -30587.462} C_VEL
LIN {X 0,Y 78.489,Z 746.117,A -85,B 0,C 180,E1 -30590.019,E2 -30590.019} C_VEL
LIN {X 0,Y 88.709,Z 736.974,A -85,B 0,C 180,E1 -30591.987,E2 -30591.987} C_VEL
LIN {X 0,Y 97.289,Z 727.46,A -85,B 0,C 180,E1 -30593.319,E2 -30593.319} C_VEL
LIN {X 0,Y 105.057,Z 716.897,A -85,B 0,C 180,E1 -30594.283,E2 -30594.283} C_VEL
LIN {X 0,Y 111.108,Z 706.697,A -85,B 0,C 180,E1 -30594.991,E2 -30594.991} C_VEL
LIN {X 0,Y 116.607,Z 694.932,A -85,B 0,C 180,E1 -30595.582,E2 -30595.582} C_VEL
LIN {X 0,Y 120.89,Z 682.461,A -85,B 0,C 180,E1 -30596.107,E2 -30596.107} C_VEL
LIN {X 0,Y 121.088,Z 681.033,A -85,B 0,C 180,E1 -30600,E2 -30600} C_VEL
LIN {X 0,Y 120.979,Z 682.37,A -85,B 0,C 180,E1 -30603.445,E2 -30603.445} C_VEL
LIN {X 0,Y 117.453,Z 693.021,A -85,B 0,C 180,E1 -30603.858,E2 -30603.858} C_VEL
LIN {X 0,Y 111.87,Z 705.552,A -85,B 0,C 180,E1 -30604.252,E2 -30604.252} C_VEL
LIN {X 0,Y 104.923,Z 717.447,A -85,B 0,C 180,E1 -30604.933,E2 -30604.933} C_VEL
LIN {X 0,Y 97.116,Z 728.057,A -85,B 0,C 180,E1 -30605.747,E2 -30605.747} C_VEL
LIN {X 0,Y 88.481,Z 737.628,A -85,B 0,C 180,E1 -30606.883,E2 -30606.883} C_VEL
LIN {X 0,Y 78.18,Z 746.838,A -85,B 0,C 180,E1 -30608.597,E2 -30608.597} C_VEL
LIN {X 0,Y 67.992,Z 754.254,A -85,B 0,C 180,E1 -30610.927,E2 -30610.927} C_VEL
LIN {X 0,Y 57.979,Z 760.213,A -85,B 0,C 180,E1 -30614.161,E2 -30614.161} C_VEL
LIN {X 0,Y 48.2,Z 764.923,A -85,B 0,C 180,E1 -30618.625,E2 -30618.625} C_VEL
LIN {X 0,Y 38.842,Z 768.529,A -85,B 0,C 180,E1 -30625.242,E2 -30625.242} C_VEL
LIN {X 0,Y 32.987,Z 770.386,A -85,B 0,C 180,E1 -30631.568,E2 -30631.568} C_VEL
LIN {X 0,Y 27.786,Z 771.785,A -85,B 0,C 180,E1 -30640.663,E2 -30640.663} C_VEL
LIN {X 0,Y 20.743,Z 773.401,A -85,B 0,C 180,E1 -30670.215,E2 -30670.215} C_VEL
LIN {X 0,Y 20.016,Z 773.618,A -85,B 0,C 180,E1 -30690.018,E2 -30690.018} C_VEL
LIN {X 0,Y 21.221,Z 773.392,A -85,B 0,C 180,E1 -30709.359,E2 -30709.359} C_VEL
LIN {X 0,Y 28.767,Z 771.771,A -85,B 0,C 180,E1 -30737.151,E2 -30737.151} C_VEL
LIN {X 0,Y 34.115,Z 770.366,A -85,B 0,C 180,E1 -30745.51,E2 -30745.51} C_VEL
LIN {X 0,Y 40.035,Z 768.502,A -85,B 0,C 180,E1 -30751.388,E2 -30751.388} C_VEL
LIN {X 0,Y 40.487,Z 767.499,A -85,B 0,C 180,E1 -30759.686,E2 -30759.686} C_VEL
LIN {X 0,Y 50.126,Z 763.1,A -85,B 0,C 180,E1 -30798.103,E2 -30798.103} C_VEL
LIN {X 0,Y 47.825,Z 764.262,A -85,B 0,C 180,E1 -30800.942,E2 -30800.942} C_VEL
LIN {X 0,Y 39.489,Z 767.425,A -85,B 0,C 180,E1 -30807.123,E2 -30807.123} C_VEL
LIN {X 0,Y 33.708,Z 769.27,A -85,B 0,C 180,E1 -30813.471,E2 -30813.471} C_VEL
LIN {X 0,Y 24.16,Z 771.635,A -85,B 0,C 180,E1 -30834.406,E2 -30834.406} C_VEL
LIN {X 0,Y 20.214,Z 772.458,A -85,B 0,C 180,E1 -30869.982,E2 -30869.982} C_VEL
LIN {X 0,Y 21.182,Z 772.263,A -85,B 0,C 180,E1 -30889.359,E2 -30889.359} C_VEL
LIN {X 0,Y 24.152,Z 771.678,A -85,B 0,C 180,E1 -30905.571,E2 -30905.571} C_VEL
LIN {X 0,Y 33.688,Z 769.355,A -85,B 0,C 180,E1 -30926.541,E2 -30926.541} C_VEL
LIN {X 0,Y 42.464,Z 766.483,A -85,B 0,C 180,E1 -30935.521,E2 -30935.521} C_VEL
LIN {X 0,Y 51.915,Z 762.582,A -85,B 0,C 180,E1 -30941.35,E2 -30941.35} C_VEL
LIN {X 0,Y 57.527,Z 759.812,A -85,B 0,C 180,E1 -30943.796,E2 -30943.796} C_VEL
LIN {X 0,Y 62.244,Z 757.218,A -85,B 0,C 180,E1 -30946.145,E2 -30946.145} C_VEL
LIN {X 0,Y 69.31,Z 752.624,A -85,B 0,C 180,E1 -30950.735,E2 -30950.735} C_VEL
LIN {X 0,Y 76.31,Z 747.38,A -85,B 0,C 180,E1 -30954.47,E2 -30954.47} C_VEL
LIN {X 0,Y 80.716,Z 743.766,A -85,B 0,C 180,E1 -30955.656,E2 -30955.656} C_VEL
LIN {X 0,Y 89.742,Z 735.401,A -85,B 0,C 180,E1 -30956.771,E2 -30956.771} C_VEL
LIN {X 0,Y 98.468,Z 725.528,A -85,B 0,C 180,E1 -30957.644,E2 -30957.644} C_VEL
LIN {X 0,Y 106.337,Z 714.401,A -85,B 0,C 180,E1 -30958.326,E2 -30958.326} C_VEL
LIN {X 0,Y 113.166,Z 702.078,A -85,B 0,C 180,E1 -30958.797,E2 -30958.797} C_VEL
LIN {X 0,Y 118.397,Z 689.57,A -85,B 0,C 180,E1 -30959.246,E2 -30959.246} C_VEL
LIN {X 0,Y 118.93,Z 687.988,A -85,B 0,C 180,E1 -30959.577,E2 -30959.577} C_VEL
LIN {X 0,Y 118.954,Z 687.931,A -85,B 0,C 180,E1 -30960,E2 -30960} C_VEL
LIN {X 0,Y 118.664,Z 688.81,A -85,B 0,C 180,E1 -30960.281,E2 -30960.281} C_VEL
LIN {X 0,Y 113.846,Z 700.741,A -85,B 0,C 180,E1 -30960.529,E2 -30960.529} C_VEL
LIN {X 0,Y 108.059,Z 711.682,A -85,B 0,C 180,E1 -30960.82,E2 -30960.82} C_VEL
LIN {X 0,Y 100.168,Z 723.423,A -85,B 0,C 180,E1 -30961.319,E2 -30961.319} C_VEL
LIN {X 0,Y 91.409,Z 733.847,A -85,B 0,C 180,E1 -30961.932,E2 -30961.932} C_VEL
LIN {X 0,Y 82.67,Z 742.291,A -85,B 0,C 180,E1 -30962.789,E2 -30962.789} C_VEL
LIN {X 0,Y 72.213,Z 750.541,A -85,B 0,C 180,E1 -30964.081,E2 -30964.081} C_VEL
LIN {X 0,Y 61.818,Z 757.197,A -85,B 0,C 180,E1 -30965.936,E2 -30965.936} C_VEL
LIN {X 0,Y 49.824,Z 763.285,A -85,B 0,C 180,E1 -30969.157,E2 -30969.157} C_VEL
LIN {X 0,Y 39.695,Z 767.248,A -85,B 0,C 180,E1 -30973.193,E2 -30973.193} C_VEL
LIN {X 0,Y 29.879,Z 770.181,A -85,B 0,C 180,E1 -30979.839,E2 -30979.839} C_VEL
LIN {X 0,Y 18.302,Z 772.581,A -85,B 0,C 180,E1 -30999.856,E2 -30999.856} C_VEL
LIN {X 0,Y 14.247,Z 773.195,A -85,B 0,C 180,E1 -31020.472,E2 -31020.472} C_VEL
LIN {X 0,Y 12.923,Z 773.413,A -85,B 0,C 180,E1 -31050.028,E2 -31050.028} C_VEL
LIN {X 0,Y 14.728,Z 773.188,A -85,B 0,C 180,E1 -31078.53,E2 -31078.53} C_VEL
LIN {X 0,Y 24.497,Z 771.566,A -85,B 0,C 180,E1 -31109.423,E2 -31109.423} C_VEL
LIN {X 0,Y 32.552,Z 769.639,A -85,B 0,C 180,E1 -31118.024,E2 -31118.024} C_VEL
LIN {X 0,Y 33.66,Z 769.04,A -85,B 0,C 180,E1 -31123.387,E2 -31123.387} C_VEL
LIN {X 0,Y 39.525,Z 766.673,A -85,B 0,C 180,E1 -31153.107,E2 -31153.107} C_VEL
LIN {X 0,Y 36.797,Z 767.631,A -85,B 0,C 180,E1 -31157.228,E2 -31157.228} C_VEL
LIN {X 0,Y 30.37,Z 769.476,A -85,B 0,C 180,E1 -31162.201,E2 -31162.201} C_VEL
LIN {X 0,Y 18.843,Z 771.841,A -85,B 0,C 180,E1 -31181.73,E2 -31181.73} C_VEL
LIN {X 0,Y 14.699,Z 772.442,A -85,B 0,C 180,E1 -31201.409,E2 -31201.409} C_VEL
LIN {X 0,Y 13.126,Z 772.662,A -85,B 0,C 180,E1 -31229.972,E2 -31229.972} C_VEL
LIN {X 0,Y 14.692,Z 772.467,A -85,B 0,C 180,E1 -31258.55,E2 -31258.55} C_VEL
LIN {X 0,Y 18.833,Z 771.882,A -85,B 0,C 180,E1 -31278.247,E2 -31278.247} C_VEL
LIN {X 0,Y 30.35,Z 769.56,A -85,B 0,C 180,E1 -31297.825,E2 -31297.825} C_VEL
LIN {X 0,Y 40.045,Z 766.687,A -85,B 0,C 180,E1 -31304.816,E2 -31304.816} C_VEL
LIN {X 0,Y 50.101,Z 762.785,A -85,B 0,C 180,E1 -31309.053,E2 -31309.053} C_VEL
LIN {X 0,Y 60.341,Z 757.753,A -85,B 0,C 180,E1 -31311.849,E2 -31311.849} C_VEL
LIN {X 0,Y 70.666,Z 751.413,A -85,B 0,C 180,E1 -31313.956,E2 -31313.956} C_VEL
LIN {X 0,Y 80.716,Z 743.766,A -85,B 0,C 180,E1 -31315.656,E2 -31315.656} C_VEL
LIN {X 0,Y 80.065,Z 744.295,A -85,B 0,C 180,E1 -31316.276,E2 -31316.276} C_VEL
LIN {X 0,Y 76.575,Z 747.071,A -85,B 0,C 180,E1 -31317.236,E2 -31317.236} C_VEL
LIN {X 0,Y 69.152,Z 752.327,A -85,B 0,C 180,E1 -31318.283,E2 -31318.283} C_VEL
LIN {X 0,Y 59.161,Z 758.281,A -85,B 0,C 180,E1 -31319.545,E2 -31319.545} C_VEL
LIN {X 0,Y 53.97,Z 760.903,A -85,B 0,C 180,E1 -31320.207,E2 -31320.207} C_VEL
LIN {X 0,Y 42.188,Z 765.821,A -85,B 0,C 180,E1 -31322.035,E2 -31322.035} C_VEL
LIN {X 0,Y 35.21,Z 768.119,A -85,B 0,C 180,E1 -31323.774,E2 -31323.774} C_VEL
LIN {X 0,Y 28.267,Z 769.976,A -85,B 0,C 180,E1 -31326.127,E2 -31326.127} C_VEL
LIN {X 0,Y 14.784,Z 772.376,A -85,B 0,C 180,E1 -31338.131,E2 -31338.131} C_VEL
LIN {X 0,Y 8.789,Z 772.991,A -85,B 0,C 180,E1 -31356.975,E2 -31356.975} C_VEL
LIN {X 0,Y 5.817,Z 773.208,A -85,B 0,C 180,E1 -31410.062,E2 -31410.062} C_VEL
LIN {X 0,Y 9.16,Z 772.984,A -85,B 0,C 180,E1 -31460.17,E2 -31460.17} C_VEL
LIN {X 0,Y 21.763,Z 771.361,A -85,B 0,C 180,E1 -31485.719,E2 -31485.719} C_VEL
LIN {X 0,Y 25.161,Z 770.695,A -85,B 0,C 180,E1 -31487.928,E2 -31487.928} C_VEL
LIN {X 0,Y 27.244,Z 770.146,A -85,B 0,C 180,E1 -31492.597,E2 -31492.597} C_VEL
LIN {X 0,Y 28.247,Z 769.777,A -85,B 0,C 180,E1 -31500.001,E2 -31500.001} C_VEL
LIN {X 0,Y 28.454,Z 769.682,A -85,B 0,C 180,E1 -31508.816,E2 -31508.816} C_VEL
LIN {X 0,Y 15.081,Z 772.045,A -85,B 0,C 180,E1 -31521.181,E2 -31521.181} C_VEL
LIN {X 0,Y 9.125,Z 772.647,A -85,B 0,C 180,E1 -31539.568,E2 -31539.568} C_VEL
LIN {X 0,Y 6.027,Z 772.867,A -85,B 0,C 180,E1 -31589.94,E2 -31589.94} C_VEL
LIN {X 0,Y 9.115,Z 772.671,A -85,B 0,C 180,E1 -31640.386,E2 -31640.386} C_VEL
LIN {X 0,Y 15.069,Z 772.087,A -85,B 0,C 180,E1 -31658.806,E2 -31658.806} C_VEL
LIN {X 0,Y 28.438,Z 769.765,A -85,B 0,C 180,E1 -31671.225,E2 -31671.225} C_VEL
LIN {X 0,Y 38.793,Z 766.891,A -85,B 0,C 180,E1 -31675.03,E2 -31675.03} C_VEL
LIN {X 0,Y 51.473,Z 762.006,A -85,B 0,C 180,E1 -31677.576,E2 -31677.576} C_VEL
LIN {X 0,Y 63.253,Z 755.977,A -85,B 0,C 180,E1 -31679.075,E2 -31679.075} C_VEL
LIN {X 0,Y 53.97,Z 760.903,A -85,B 0,C 180,E1 -31680.207,E2 -31680.207} C_VEL
LIN {X 0,Y 53.97,Z 760.903,A -85,B 0,C 180,E1 -31680.207,E2 -31680.207}

QRS_NEXT_CUT()

QRS_NEXT()
QRS_HOME()

END
